TYPE ST_InfoDataFB :
STRUCT
	usiMapState:USINT;
	uiMapDiag:USINT;
	usiDummy:USINT;
END_STRUCT
END_TYPE

(* stored: Version 1.1.0.1, ProductVersion 3.1.0.20
   DUT ST_InfoDataFB: Id {f292264d-0e04-4f99-9d1d-065f4d7dd942} *)
